FUNCTION_BLOCK BaseState IMPLEMENTS itfState
VAR_INPUT
	BasePointer : POINTER TO WRAPPER;
END_VAR
VAR_OUTPUT
END_VAR
VAR
	StateTimer : TON;
	Index : INT;
	TESTING : INT;
END_VAR

METHOD FB_INIT : BOOL
VAR_INPUT
	bInitRetains : BOOL;
	bInCopyCode : BOOL;
	WrapperPointer : POINTER TO Wrapper;
END_VAR
BasePointer := WrapperPointer;
END_METHOD

METHOD PROTECTED mCheckDosing : BOOL
VAR_INPUT
END_VAR
FOR INDEX :=1 TO BasePointer^.pNUM_SILOS BY 1 DO
	IF BasePointer^.SpiralAccessI[INDEX].mRunning() THEN
		RETURN;
	END_IF
END_FOR

mCheckDosing := TRUE;
END_METHOD

METHOD mIrun : BOOL
END_METHOD

METHOD mNextState : BOOL
VAR_INPUT
END_VAR
StateTimer(IN:= TRUE, PT:= T#1000MS);

IF StateTimer.Q THEN
BasePointer^.pStateIndex := BasePointer^.pStateIndex + 1;
StateTimer(IN:= FALSE);
END_IF
END_METHOD

END_FUNCTION_BLOCK

(* stored: Version 1.1.0.1, ProductVersion 3.1.4024.12
   POU BaseState: Id {2b11ec1c-7853-4863-bf5c-bd9acf84bec2}, SpecialFunc None
   Method FB_INIT: Id {529836ac-3a75-43d8-b9ff-70a071d414a1}
   Method mCheckDosing: Id {e93c066a-1ad2-4525-a6e4-24a2d19d5695}
   Method mIrun: Id {9c8d0b80-7873-4ac4-b5d7-be821cca1725}
   Method mNextState: Id {dfaa6ff3-2f6a-45d4-b276-b711de275c3b} *)
